DATA_BLOCK "DB3_C"
{ S7_Optimized_Access := 'TRUE' }
NAME : FCDI
VERSION : 0.1
NON_RETAIN
"FB2_C"

BEGIN
   increment_C := 111444;
   counter_C := 92146;
   dnCALLCHECK_C := 87957;
   dnTRACER_START := 20944;
   dnGCTX_DBNUMBER := 30011;

END_DATA_BLOCK

